{attribute 'strict'}
TYPE E_SMStatus :
(Initialize,
Read,
SystemCheck,
Automatic,
Write,
Error);
END_TYPE

(* stored: Version 1.1.0.1, ProductVersion 3.1.4018.2
   DUT E_SMStatus: Id {3c99a96b-f127-4015-9b5f-06a7e2b7a393} *)
